// TIA Portal V19 export
FUNCTION_BLOCK "Straightener_FB"   // FB44, LAD
TITLE = STRAIGHTENER
// stored: MemoryReserve 100, SetENOAutomatically false
   VAR_INPUT
      AreaInterface : "AreaInterface";
      ZSI : "udt_ZoneSafetyInterface";
      DSI : Struct
         Feed : "udt_DeviceSafetyInterface";
         Lift_Entry : "udt_DeviceSafetyInterface";
         Lift_Exit : "udt_DeviceSafetyInterface";
      END_STRUCT;
      Drive : Struct
         Feed : "TAx_DriveInterface";
      END_STRUCT;
      DataIn : Struct
         Feed : "PositioningMachine_DataIn";
         Lift_Entry : "ValveMachine_DataIn";
         Lift_Exit : "ValveMachine_DataIn";
      END_STRUCT;
      CIn : Struct
         Manager : "Straightener_Manager";
         Feed_BwdEnable : Array[1..8] of Bool;
         Feed_FwdEnable : Array[1..8] of Bool;
      END_STRUCT;
      Config : Struct
         Feed : "PositioningMachine_Config";
         Lift_Entry : "ValveMachine_Config";
         Lift_Exit : "ValveMachine_Config";
         Lift_Entry_Exist : Bool;
         Lift_Exit_Exist : Bool;
      END_STRUCT;
   END_VAR
   VAR_OUTPUT
      MachineInterface : "MachineInterface";
      DataOut : Struct
         Feed : "PositioningMachine_DataOut";
         Lift_Entry : "ValveMachine_DataOut";
         Lift_Exit : "ValveMachine_DataOut";
      END_STRUCT;
      COut : "Straightener_Status";
   END_VAR
   VAR_IN_OUT
      TO_Ax : TO_PositioningAxis;
      PersistentValues : Struct
         Data : Struct
            Feed : "PositioningMachine_DataPers";
         END_STRUCT;
         Feed : "PositioningMachine_Par";
      END_STRUCT;
   END_VAR
   VAR
      Alarm : Struct
         Feed : "PositioningMachine_Alr";
         Lift_Entry : "ValveAlr";
         Lift_Exit : "ValveAlr";
      END_STRUCT;
      Warning : Struct
         Feed : "PositioningMachine_Wng";
         Lift_Entry : "ValveMachine_Wng";
         Lift_Exit : "ValveMachine_Wng";
      END_STRUCT;
      Feed : "PositioningMachine_FB";
      Lift_Entry : "ValveMachine_FB";
      Lift_Exit : "ValveMachine_FB";
   END_VAR
   VAR_TEMP
      ExternalWorkCmd : Bool;
      InternalWorkCmd : Bool;
      ExternalRestEnable : Bool;
      InternalRestEnable : Bool;
      ExternaleWorkEnable : Bool;
      InternalWorkEnable : Bool;
   END_VAR
BEGIN

REGION Network 1: <<< FEED >>>
END_REGION

REGION Network 2: CIn (External Bwd / Fwd enable)
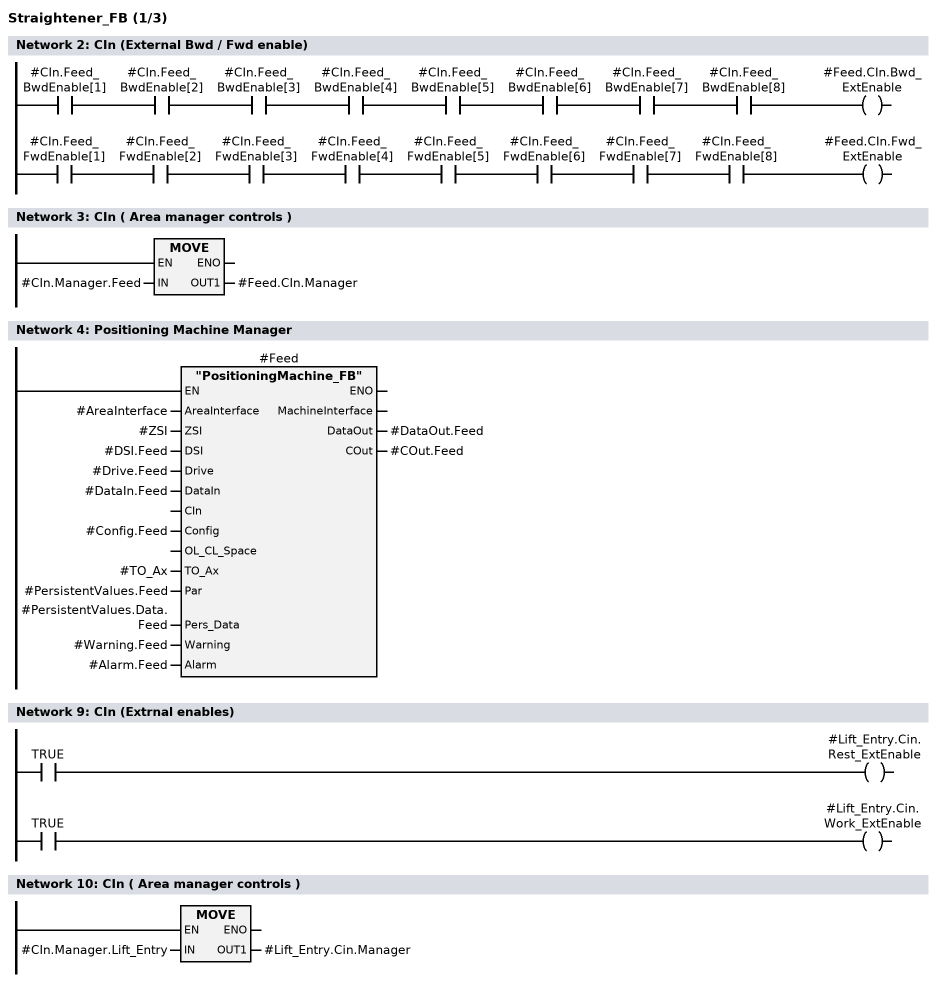
   RUNG wire#powerrail
      Contact( #CIn.Feed_BwdEnable[1] )
      Contact( #CIn.Feed_BwdEnable[2] )
      Contact( #CIn.Feed_BwdEnable[3] )
      Contact( #CIn.Feed_BwdEnable[4] )
      Contact( #CIn.Feed_BwdEnable[5] )
      Contact( #CIn.Feed_BwdEnable[6] )
      Contact( #CIn.Feed_BwdEnable[7] )
      Contact( #CIn.Feed_BwdEnable[8] )
      Coil( #Feed.CIn.Bwd_ExtEnable )
   END_RUNG
   RUNG wire#powerrail
      Contact( #CIn.Feed_FwdEnable[1] )
      Contact( #CIn.Feed_FwdEnable[2] )
      Contact( #CIn.Feed_FwdEnable[3] )
      Contact( #CIn.Feed_FwdEnable[4] )
      Contact( #CIn.Feed_FwdEnable[5] )
      Contact( #CIn.Feed_FwdEnable[6] )
      Contact( #CIn.Feed_FwdEnable[7] )
      Contact( #CIn.Feed_FwdEnable[8] )
      Coil( #Feed.CIn.Fwd_ExtEnable )
   END_RUNG
   // the same network as SCL:
   #Feed.CIn.Bwd_ExtEnable := #CIn.Feed_BwdEnable[1] AND #CIn.Feed_BwdEnable[2] AND #CIn.Feed_BwdEnable[3] AND #CIn.Feed_BwdEnable[4] AND #CIn.Feed_BwdEnable[5] AND #CIn.Feed_BwdEnable[6] AND #CIn.Feed_BwdEnable[7] AND #CIn.Feed_BwdEnable[8];
   #Feed.CIn.Fwd_ExtEnable := #CIn.Feed_FwdEnable[1] AND #CIn.Feed_FwdEnable[2] AND #CIn.Feed_FwdEnable[3] AND #CIn.Feed_FwdEnable[4] AND #CIn.Feed_FwdEnable[5] AND #CIn.Feed_FwdEnable[6] AND #CIn.Feed_FwdEnable[7] AND #CIn.Feed_FwdEnable[8];
END_REGION

REGION Network 3: CIn ( Area manager controls )
   RUNG wire#powerrail
      { S7_GenerateENO := "TRUE" } Move(in := #CIn.Manager.Feed, out1 => #Feed.CIn.Manager)
   END_RUNG
   // the same network as SCL:
   #Feed.CIn.Manager := #CIn.Manager.Feed;
END_REGION

REGION Network 4: Positioning Machine Manager
   RUNG wire#powerrail
      #Feed(AreaInterface := #AreaInterface, ZSI := #ZSI, DSI := #DSI.Feed, Drive := #Drive.Feed, DataIn := #DataIn.Feed, CIn :=, Config := #Config.Feed, OL_CL_Space :=, TO_Ax := #TO_Ax, Par := #PersistentValues.Feed, Pers_Data := #PersistentValues.Data.Feed, Warning := #Warning.Feed, Alarm := #Alarm.Feed, MachineInterface =>, DataOut => #DataOut.Feed, COut => #COut.Feed)
   END_RUNG
   // the same network as SCL:
   #Feed(AreaInterface := #AreaInterface,   // "PositioningMachine_FB"
         ZSI := #ZSI,
         DSI := #DSI.Feed,
         Drive := #Drive.Feed,
         DataIn := #DataIn.Feed,
         Config := #Config.Feed,
         TO_Ax := #TO_Ax,
         Par := #PersistentValues.Feed,
         Pers_Data := #PersistentValues.Data.Feed,
         Warning := #Warning.Feed,
         Alarm := #Alarm.Feed,
         DataOut => #DataOut.Feed,
         COut => #COut.Feed);
END_REGION

REGION Network 6: >
END_REGION

REGION Network 7: >
END_REGION

REGION Network 8: <<< LIFT ENTRY >>>
END_REGION

REGION Network 9: CIn (Extrnal enables)
   RUNG wire#powerrail
      Contact( TRUE )
      Coil( #Lift_Entry.Cin.Rest_ExtEnable )
   END_RUNG
   RUNG wire#powerrail
      Contact( TRUE )
      Coil( #Lift_Entry.Cin.Work_ExtEnable )
   END_RUNG
   // the same network as SCL:
   #Lift_Entry.Cin.Rest_ExtEnable := TRUE;
   #Lift_Entry.Cin.Work_ExtEnable := TRUE;
END_REGION

REGION Network 10: CIn ( Area manager controls )
   RUNG wire#powerrail
      { S7_GenerateENO := "TRUE" } Move(in := #CIn.Manager.Lift_Entry, out1 => #Lift_Entry.Cin.Manager)
   END_RUNG
   // the same network as SCL:
   #Lift_Entry.Cin.Manager := #CIn.Manager.Lift_Entry;
END_REGION

REGION Network 11: Valve machine Manager
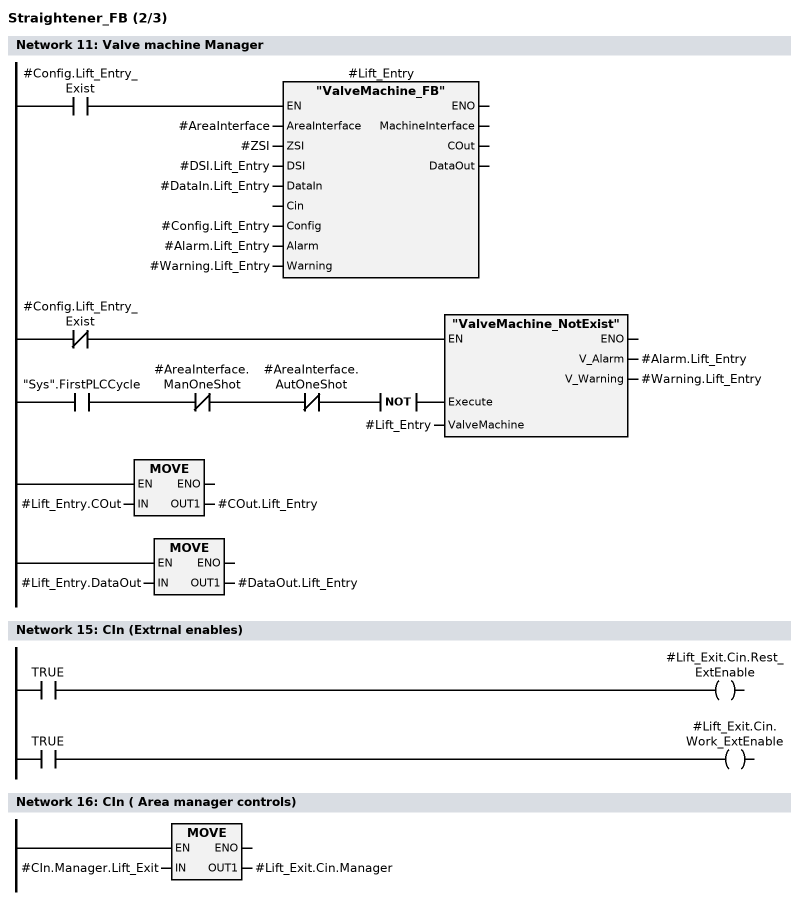
   RUNG wire#powerrail
      Contact( #Config.Lift_Entry_Exist )
      #Lift_Entry(AreaInterface := #AreaInterface, ZSI := #ZSI, DSI := #DSI.Lift_Entry, DataIn := #DataIn.Lift_Entry, Cin :=, Config := #Config.Lift_Entry, Alarm := #Alarm.Lift_Entry, Warning := #Warning.Lift_Entry, MachineInterface =>, COut =>, DataOut =>)
   END_RUNG
   RUNG wire#powerrail
      I_Contact( #Config.Lift_Entry_Exist )
      "ValveMachine_NotExist"(Execute := wire#w1, ValveMachine := #Lift_Entry, V_Alarm => #Alarm.Lift_Entry, V_Warning => #Warning.Lift_Entry)
   END_RUNG
   RUNG wire#powerrail
      Contact( "Sys".FirstPLCCycle )
      I_Contact( #AreaInterface.ManOneShot )
      I_Contact( #AreaInterface.AutOneShot )
      Not()
   END_RUNG wire#w1
   RUNG wire#powerrail
      Move(in := #Lift_Entry.COut, out1 => #COut.Lift_Entry)
   END_RUNG
   RUNG wire#powerrail
      Move(in := #Lift_Entry.DataOut, out1 => #DataOut.Lift_Entry)
   END_RUNG
   // the same network as SCL:
   IF #Config.Lift_Entry_Exist THEN
       #Lift_Entry(AreaInterface := #AreaInterface,   // "ValveMachine_FB"
                   ZSI := #ZSI,
                   DSI := #DSI.Lift_Entry,
                   DataIn := #DataIn.Lift_Entry,
                   Config := #Config.Lift_Entry,
                   Alarm := #Alarm.Lift_Entry,
                   Warning := #Warning.Lift_Entry);
   END_IF;
   IF NOT #Config.Lift_Entry_Exist THEN
       "ValveMachine_NotExist"(Execute := NOT ("Sys".FirstPLCCycle AND NOT #AreaInterface.ManOneShot AND NOT #AreaInterface.AutOneShot),
                               ValveMachine := #Lift_Entry,
                               V_Alarm => #Alarm.Lift_Entry,
                               V_Warning => #Warning.Lift_Entry);
   END_IF;
   #COut.Lift_Entry := #Lift_Entry.COut;
   #DataOut.Lift_Entry := #Lift_Entry.DataOut;
END_REGION

REGION Network 12: >
END_REGION

REGION Network 13: >
END_REGION

REGION Network 14: <<< LIFT EXIT >>>
END_REGION

REGION Network 15: CIn (Extrnal enables)
   RUNG wire#powerrail
      Contact( TRUE )
      Coil( #Lift_Exit.Cin.Rest_ExtEnable )
   END_RUNG
   RUNG wire#powerrail
      Contact( TRUE )
      Coil( #Lift_Exit.Cin.Work_ExtEnable )
   END_RUNG
   // the same network as SCL:
   #Lift_Exit.Cin.Rest_ExtEnable := TRUE;
   #Lift_Exit.Cin.Work_ExtEnable := TRUE;
END_REGION

REGION Network 16: CIn ( Area manager controls)
   RUNG wire#powerrail
      { S7_GenerateENO := "TRUE" } Move(in := #CIn.Manager.Lift_Exit, out1 => #Lift_Exit.Cin.Manager)
   END_RUNG
   // the same network as SCL:
   #Lift_Exit.Cin.Manager := #CIn.Manager.Lift_Exit;
END_REGION

REGION Network 17: Valve machine Manager
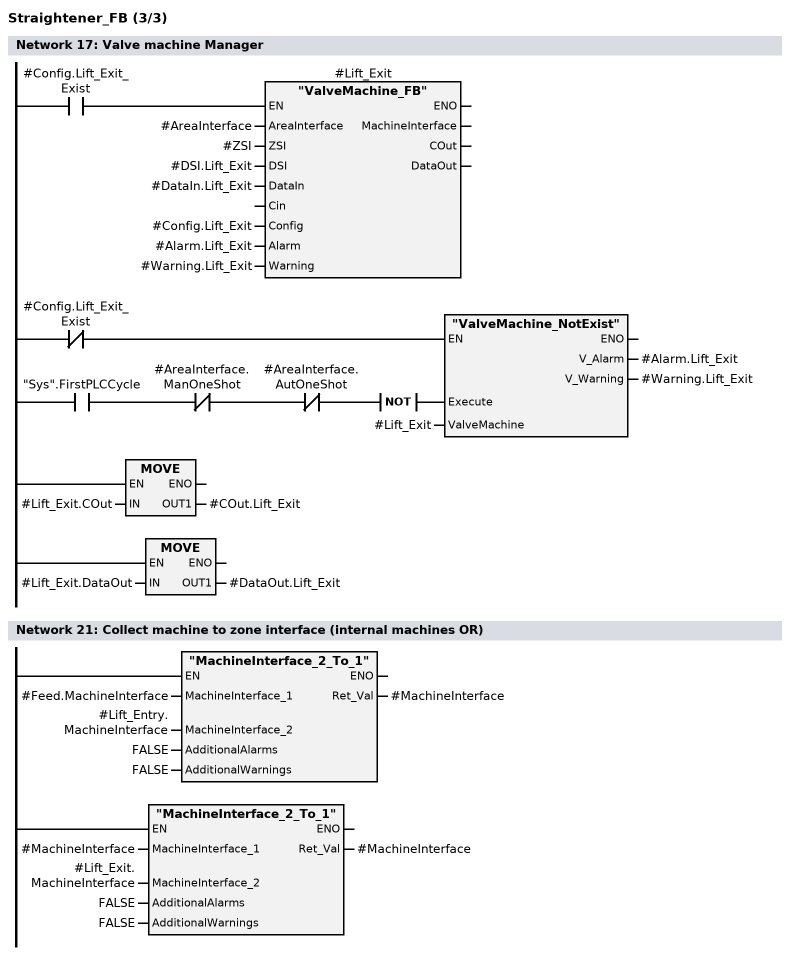
   RUNG wire#powerrail
      Contact( #Config.Lift_Exit_Exist )
      #Lift_Exit(AreaInterface := #AreaInterface, ZSI := #ZSI, DSI := #DSI.Lift_Exit, DataIn := #DataIn.Lift_Exit, Cin :=, Config := #Config.Lift_Exit, Alarm := #Alarm.Lift_Exit, Warning := #Warning.Lift_Exit, MachineInterface =>, COut =>, DataOut =>)
   END_RUNG
   RUNG wire#powerrail
      I_Contact( #Config.Lift_Exit_Exist )
      "ValveMachine_NotExist"(Execute := wire#w1, ValveMachine := #Lift_Exit, V_Alarm => #Alarm.Lift_Exit, V_Warning => #Warning.Lift_Exit)
   END_RUNG
   RUNG wire#powerrail
      Contact( "Sys".FirstPLCCycle )
      I_Contact( #AreaInterface.ManOneShot )
      I_Contact( #AreaInterface.AutOneShot )
      Not()
   END_RUNG wire#w1
   RUNG wire#powerrail
      Move(in := #Lift_Exit.COut, out1 => #COut.Lift_Exit)
   END_RUNG
   RUNG wire#powerrail
      Move(in := #Lift_Exit.DataOut, out1 => #DataOut.Lift_Exit)
   END_RUNG
   // the same network as SCL:
   IF #Config.Lift_Exit_Exist THEN
       #Lift_Exit(AreaInterface := #AreaInterface,   // "ValveMachine_FB"
                  ZSI := #ZSI,
                  DSI := #DSI.Lift_Exit,
                  DataIn := #DataIn.Lift_Exit,
                  Config := #Config.Lift_Exit,
                  Alarm := #Alarm.Lift_Exit,
                  Warning := #Warning.Lift_Exit);
   END_IF;
   IF NOT #Config.Lift_Exit_Exist THEN
       "ValveMachine_NotExist"(Execute := NOT ("Sys".FirstPLCCycle AND NOT #AreaInterface.ManOneShot AND NOT #AreaInterface.AutOneShot),
                               ValveMachine := #Lift_Exit,
                               V_Alarm => #Alarm.Lift_Exit,
                               V_Warning => #Warning.Lift_Exit);
   END_IF;
   #COut.Lift_Exit := #Lift_Exit.COut;
   #DataOut.Lift_Exit := #Lift_Exit.DataOut;
END_REGION

REGION Network 18: >
END_REGION

REGION Network 19: >
END_REGION

REGION Network 20: <<< MACHINE STATUS >>>
END_REGION

REGION Network 21: Collect machine to zone interface (internal machines OR)
   RUNG wire#powerrail
      "MachineInterface_2_To_1"(MachineInterface_1 := #Feed.MachineInterface, MachineInterface_2 := #Lift_Entry.MachineInterface, AdditionalAlarms := FALSE, AdditionalWarnings := FALSE, Ret_Val => #MachineInterface)
   END_RUNG
   RUNG wire#powerrail
      "MachineInterface_2_To_1"(MachineInterface_1 := #MachineInterface, MachineInterface_2 := #Lift_Exit.MachineInterface, AdditionalAlarms := FALSE, AdditionalWarnings := FALSE, Ret_Val => #MachineInterface)
   END_RUNG
   // the same network as SCL:
   #MachineInterface := "MachineInterface_2_To_1"(MachineInterface_1 := #Feed.MachineInterface,
                           MachineInterface_2 := #Lift_Entry.MachineInterface,
                           AdditionalAlarms := FALSE,
                           AdditionalWarnings := FALSE);
   #MachineInterface := "MachineInterface_2_To_1"(MachineInterface_1 := #MachineInterface,
                           MachineInterface_2 := #Lift_Exit.MachineInterface,
                           AdditionalAlarms := FALSE,
                           AdditionalWarnings := FALSE);
END_REGION

REGION Network 22: >
END_REGION
END_FUNCTION_BLOCK
